Omron Sysmac Studio project ToggleButton_Karsilastirma (Sysmac Studio 1.65.0.64007, StandardProject)

# Controller new_Controller_0: NX1P2-1040DT1 version 1.69
Task PrimaryTask (priority 4, period or condition 2000): Program0



PROGRAM Program0
VAR
    ToggleButton : BOOL;
    ToggleSayac : INT;
    MotorCikis : BOOL;
    MotorStart : BOOL;
END_VAR

(* Section Section0: ladder, written here as Structured Text *)

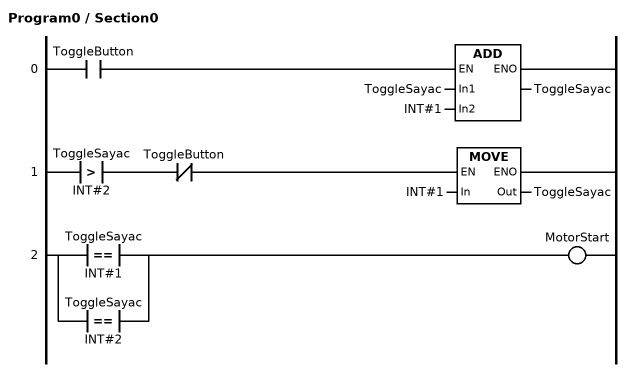
(* Rung 0 *)
IF ToggleButton THEN ToggleSayac := ToggleSayac + INT#1; END_IF;
(* Rung 1 *)
IF (ToggleSayac > INT#2) AND NOT ToggleButton THEN ToggleSayac := INT#1; END_IF;
(* Rung 2 *)
MotorStart := (ToggleSayac = INT#1) OR (ToggleSayac = INT#2);
END_PROGRAM